(* PLC project Unnamed, Unknown Unnamed 1 *)
(* stored: creationDateTime 2025-03-31T15:54:50, modificationDateTime 2025-04-01T15:01:08 *)

PROGRAM program0
  VAR
    DigitalRead AT %IW0 : WORD := 0;
  END_VAR
  VAR_EXTERNAL
    DigitalReadOut : WORD;
  END_VAR
  VAR
    userButton AT %IX1.0 : BOOL := 0;
  END_VAR
  VAR
    gtBool : BOOL := 0;
  END_VAR
  VAR
    myout AT %QX0.1 : BOOL := 1;
  END_VAR

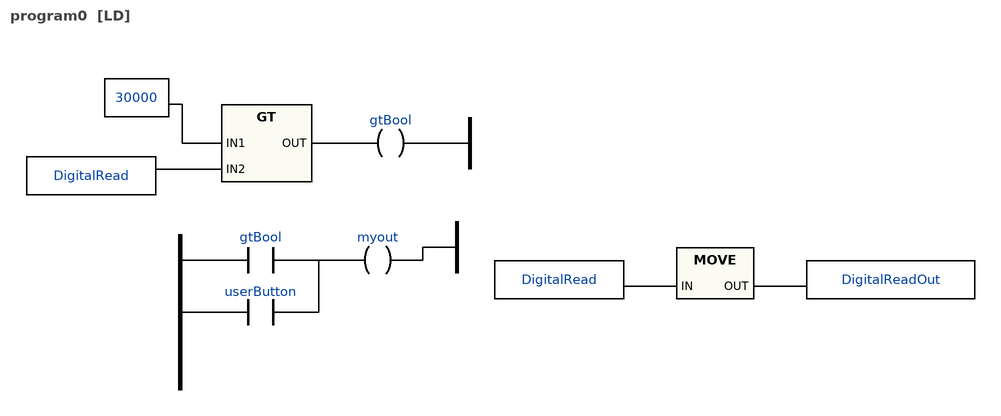
(* LD diagram, written out as Structured Text *)
gtBool := 30000 > DigitalRead;
myout := gtBool OR userButton;
DigitalReadOut := DigitalRead;
END_PROGRAM

CONFIGURATION Config0
  RESOURCE Res0 ON PLC
    TASK task0(INTERVAL := T#20ms, PRIORITY := 0);
    PROGRAM instance0 WITH task0 : program0;
  END_RESOURCE
END_CONFIGURATION
